// Core §6.8 — THE provided step-chain base: an SFC/ST/LD sequence POU extends
// this and gets the step record, condition waits, run-style pacing, the child
// PLCopen drive, delays, and the shared transition result — without re-declaring
// host plumbing per chain. The derived chart's actions are the only writers of
// _retVal; every chart transition reads it; one shared exit action calls
// M_ClearTransition. Framework flow-control lives here ONCE (§6.8(a)); the
// application's command/wait/decision logic stays visible in each step action.
FUNCTION_BLOCK ABSTRACT FB_SequenceBase IMPLEMENTS I_Sequence
VAR_OUTPUT
    ActiveStep : INT;              // §6.5 mirror of the step record (chart-local view)
    Done : BOOL;                   // finite chains: TRUE at their finish step
END_VAR
VAR
    _step    : INT;                // §6.5 active step index (the ST `CASE _step OF` token)
    // Shared transition result (§6.10). ONE-SCAN signal: the active step's action
    // is its only writer, every chart transition reads it, and it is cleared before
    // the next scan's actions run - by M_Advance on commit in an ST chart, or by
    // M_BeginScan when the chart runtime owns the transition (SFC/LD/FBD).
    _retVal  : E_StepResult;
    // §6.12 — the same one-scan signal as _retVal, but one per CONCURRENT LEG.
    // A parallel divergence has several active steps at once, so a single shared
    // result cannot work: whichever leg wrote last would decide every leg's
    // transition. Index n belongs to leg n; the main line keeps _retVal, so a
    // chain with no parallel branch never touches this array.
    //
    // A leg's step action writes `_conRetVal[n] := E_StepResult.ADVANCE;` and its
    // transition reads `_conRetVal[n] = E_StepResult.ADVANCE`; the join reads every
    // leg plus the main line. Cleared with _retVal once per scan (M_BeginScan), and
    // per leg on that leg's step exit (M_ClearTransition) - never across legs,
    // which would let one leg's commit erase another's result mid-motion.
    _conRetVal  : ARRAY[1..PL_Fraktal.MAX_PARALLEL_BRANCHES] OF E_StepResult;
    _restart : BOOL;               // a step may request a chart restart (M_Run applies it)
    {attribute 'OPC.UA.DA' := '0'}
    _host : I_SequenceHost;        // owning module's framework services (§6.7)
    _attached : BOOL;
    // §6.12 — every STEP-scoped latch is per CONCURRENT BRANCH, because two legs of
    // a parallel divergence are two active steps in the same POU at the same time.
    // Sharing one latch let leg A's issue consume leg B's, and let leg A's step exit
    // wipe leg B's transition result. Index 0 is the main line, which is what a chain
    // without any parallel branch uses throughout.
    _delay : ARRAY[0..PL_Fraktal.MAX_PARALLEL_BRANCHES] OF TON;
    _driveIssued : ARRAY[0..PL_Fraktal.MAX_PARALLEL_BRANCHES] OF BOOL;
    _subRunning : ARRAY[0..PL_Fraktal.MAX_PARALLEL_BRANCHES] OF BOOL;
    // Which leg the step action executing RIGHT NOW belongs to. Set by M_Step from
    // its `Branch` input, so it is always in step with the record just published,
    // and reset to _branchBase every scan - a chain that never names a leg is
    // therefore always on its own, which for a top-level chain is the main line.
    _branch : INT;
    // This chain's own leg index when the chain IS a leg (assigned by M_RunPar at
    // the fork). 0 for a top-level chain. It is what lets a leg written as its own
    // chain tag every one of its rows without naming a branch anywhere.
    _branchBase : INT;
    _lastStep : ARRAY[0..PL_Fraktal.MAX_PARALLEL_BRANCHES] OF INT;
    _stepSeen : ARRAY[0..PL_Fraktal.MAX_PARALLEL_BRANCHES] OF BOOL;
    _parStarted : ARRAY[1..PL_Fraktal.MAX_PARALLEL_BRANCHES] OF BOOL;
    _parLegs : INT;                // M_RunPar calls made this scan
    _parDone : INT;                // how many of them reported Done
    _errorRaised : BOOL;           // this chain raised the active fault (§6.9)
    _warnRaised : ARRAY[0..PL_Fraktal.MAX_PARALLEL_BRANCHES] OF BOOL;   // §6.9(e) one message per step visit
    _baseStepNo : INT;             // §6.5 step-record offset when run as a sub-chain
END_VAR

;

// §6.8 ST-skeleton progression: at the END of a `CASE _step OF` body, commit the
// step's shared transition result. On ADVANCE (or a declared JUMPn) go to the
// mapped next step and clear the step-scoped latches so the new step re-arms — the
// exact guarantee the SFC exit action gave, in one call. NONE stays put. The caller
// passes its successor map; an unmapped result holds the step (safe, visible).
METHOD M_Advance
VAR_INPUT
    OnAdvance : INT;               // next step for E_StepResult.ADVANCE
    // Jump targets default to "not used" so the common case reads
    // `M_Advance(OnAdvance := 100);` instead of repeating `OnJump1..3 := -1`.
    // Defaulted METHOD inputs need TwinCAT >= 3.1.4026, so on the legacy 4024
    // target (FRAKTAL_TC3_4024 defined) they are declared without defaults and
    // every argument is passed explicitly. See Params/PL_FraktalCompat.TcGVL.
    {IF defined (FRAKTAL_TC3_4024)}
    OnJump1   : INT;               // next step for JUMP1 (-1 = not used)
    OnJump2   : INT;               // next step for JUMP2 (-1 = not used)
    OnJump3   : INT;               // next step for JUMP3 (-1 = not used)
    {ELSE}
    OnJump1   : INT := -1;         // next step for JUMP1 (-1 = not used)
    OnJump2   : INT := -1;         // next step for JUMP2 (-1 = not used)
    OnJump3   : INT := -1;         // next step for JUMP3 (-1 = not used)
    {END_IF}
END_VAR
VAR
    target : INT;
END_VAR
target := -1;
CASE _retVal OF
    E_StepResult.ADVANCE: target := OnAdvance;
    E_StepResult.JUMP1:   target := OnJump1;
    E_StepResult.JUMP2:   target := OnJump2;
    E_StepResult.JUMP3:   target := OnJump3;
END_CASE
IF target >= 0 THEN
    _step := target;
    ActiveStep := target;
    M_ClearTransition();           // §6.10: a completed result never leaks into the next step
END_IF
END_METHOD

// §6.11 forward
METHOD M_AskDecision
VAR_INPUT
    Req : ST_DecisionRequest;
END_VAR
IF _host <> 0 THEN
    _host.M_SequenceAskDecision(Req := Req);
END_IF
END_METHOD

// bind the owner's host bridge; the derived Setup adds its typed child bindings.
METHOD M_Attach : BOOL
VAR_INPUT
    Host : I_SequenceHost;
END_VAR
_host := Host;
_attached := (Host <> 0);
IF _attached THEN
    // Announce this chain to its owner so the Unit base can run the
    // §6.10 per-scan result reset for it. The project writes nothing (O1).
    _host.M_SequenceRegister(Seq := THIS^);
END_IF
M_Attach := _attached;
END_METHOD

// §6.9(b) named plain-condition wait (forward to the host).
METHOD M_Await : BOOL
VAR_INPUT
    Idx : INT;
    Label : STRING(120);
    Ok : BOOL;
END_VAR
M_Await := FALSE;
IF _host <> 0 THEN
    M_Await := _host.M_SequenceAwait(Idx := Idx, Label := Label, Ok := Ok);
END_IF
END_METHOD

// Core §6.10 - scan-scoped reset of the shared transition result.
//
// `_retVal` is a ONE-SCAN signal: the active step's action writes it, the chart's
// transition reads it in the same scan, and it must not survive into the next.
// In an ST chart M_Advance is itself the transition, so it commits and clears in
// one call. In a chart language the RUNTIME evaluates transitions (SFC/LD/FBD),
// so nothing in the chart is positioned to clear afterwards - call this once per
// PLC cycle immediately BEFORE executing the chart. Clearing at the top of the
// scan is equivalent to clearing after the previous scan's transitions, and it
// forces every step action to re-assert its own result each scan, which is the
// property that makes a stale ADVANCE impossible.
//
// It deliberately clears ONLY the result. `_driveIssued` (M_TryIssue's one-shot)
// and `_delay` (M_Delay's timer) are STEP-scoped, not scan-scoped: resetting them
// every scan would re-issue a child command every cycle and stop any delay from
// ever elapsing. Those re-arm on step change, through M_ClearTransition.
METHOD M_BeginScan
VAR
	Idx : INT;
END_VAR
_retVal := E_StepResult.NONE;
FOR Idx := 1 TO PL_Fraktal.MAX_PARALLEL_BRANCHES DO
    _conRetVal[Idx] := E_StepResult.NONE;
END_FOR
// §6.12 the branch cursor is scan-scoped: a step action that does not declare a
// branch is on the main line (or on this chain's own leg when it IS a leg), so a
// chain with no parallel branch never mentions one.
_branch := _branchBase;
_parLegs := 0;
_parDone := 0;
END_METHOD

// Restart this chain as a sub-chain of a composite step: its step records are
// offset by the owning step number (§6.5) so the stall walk still reports one
// continuous chain. OnChainReset carries any application state.
METHOD M_ChainReset
VAR_INPUT
    BaseStepNo : INT;
    // §6.12 the leg index this chain runs as, assigned by the fork. 0 = not a leg.
    // Every step it records is tagged with it, so the project writes it once per
    // leg instead of once per step (§1.1 O1).
    Branch : INT;
END_VAR
_baseStepNo := BaseStepNo;
_branchBase := Branch;
M_ResetBase(FirstStep := 0);
OnChainReset();
END_METHOD

// §6.12 — the join of a parallel step: ADVANCE on the scan every leg run this
// scan has reported Done, NONE while any is still working. The counts are
// scan-scoped, so the join always reflects the legs the step actually ran -
// there is no leg list to register, and none to forget to update (§1.1 O1).
METHOD M_ParJoin : E_StepResult
M_ParJoin := E_StepResult.NONE;
IF (_parLegs > 0) AND (_parDone = _parLegs) THEN
    M_ParJoin := E_StepResult.ADVANCE;
END_IF
END_METHOD

// §6.12 — run one leg of a parallel step. THE portable form of a parallel
// divergence, and the only one available to an ST chain.
//
//     M_Step(StepNo := 500, StepName := 'project.step.bothPositions', ...);
//     M_RunPar(Chain := _positionA, BaseStepNo := 500, Branch := 1);
//     M_RunPar(Chain := _positionB, BaseStepNo := 600, Branch := 2);
//     _retVal := M_ParJoin();
//     M_Advance(OnAdvance := 999);
//
// Each leg is an ordinary FB_SequenceBase chain, so it brings its own step
// pointer, its own transition result and its own step-scoped latches - the
// collisions §6.12 has to manage inside one POU simply cannot arise (§1.1 O4:
// the model scales structurally rather than by decoration). Its steps are
// recorded under BaseStepNo and tagged with Branch, so the §3.13 flow chart
// groups them and the §6.9 walk still names one continuous chain.
//
// Returns TRUE on the scans this leg reports Done. The entry latch is
// step-scoped, so re-entering the fork step later restarts every leg.
METHOD M_RunPar : BOOL
VAR_INPUT
    Chain : REFERENCE TO FB_SequenceBase;
    BaseStepNo : INT;
    Branch : INT;
END_VAR
M_RunPar := FALSE;
IF NOT __ISVALIDREF(Chain) THEN
    RETURN;
END_IF
IF (Branch < 1) OR (Branch > PL_Fraktal.MAX_PARALLEL_BRANCHES) THEN
    M_Fault(Reason := E_Reason.UNSUPPORTED_COMMAND,
        DescriptionKey := 'std.error.parallelBranchOutOfRange');
    RETURN;                          // §5.6 no silent default
END_IF
IF NOT _parStarted[Branch] THEN
    Chain.M_ChainReset(BaseStepNo := BaseStepNo, Branch := Branch);
    _parStarted[Branch] := TRUE;
END_IF
Chain.M_ChainRun();
_parLegs := _parLegs + 1;
IF Chain.Done THEN
    _parDone := _parDone + 1;
    M_RunPar := TRUE;
END_IF
END_METHOD

// One scan of this chain. An ST chart overrides this with its
// `CASE _step OF` body; a chart-language POU leaves it alone because its own body
// IS the chart and the runtime executes it. Only a chain that is used as a
// composite step (M_RunSub) has to override it.
METHOD M_ChainRun
;
END_METHOD

METHOD M_ClearDecision
IF _host <> 0 THEN
    _host.M_SequenceClearDecision();
END_IF
END_METHOD

// the ONE shared STEP-EXIT action: a completed step's result never leaks into
// the next step, and the step-scoped helpers (delay, drive latch) re-arm.
// §6.12 — it re-arms THE CURRENT BRANCH only. Clearing every branch here is what
// made a parallel divergence misbehave: one leg committing a step wiped the other
// leg's transition result and its issue latch mid-motion.
// ST charts reach this through M_Advance on commit. A chart language whose
// engine owns the transition (SFC/LD/FBD) wires this as the step exit action,
// which the runtime executes AFTER the transition condition was evaluated -
// so the transition still sees the result the step action produced.
METHOD M_ClearTransition
VAR
	Idx : INT;
END_VAR
IF _branch = 0 THEN
    _retVal := E_StepResult.NONE;
    // A fork always sits on the main line of its own chain (§6.12), so leaving the
    // fork step is what re-arms its legs for a later re-entry.
    FOR Idx := 1 TO PL_Fraktal.MAX_PARALLEL_BRANCHES DO
        _parStarted[Idx] := FALSE;
    END_FOR
ELSE
    _conRetVal[_branch] := E_StepResult.NONE;
END_IF
_driveIssued[_branch] := FALSE;
_warnRaised[_branch] := FALSE;
_subRunning[_branch] := FALSE;
_delay[_branch](IN := FALSE);
END_METHOD

// §6.1 one-shot completion forward (finite chains)
METHOD M_Complete
IF _host <> 0 THEN
    _host.M_SequenceComplete();
END_IF
END_METHOD

METHOD M_CountGood
IF _host <> 0 THEN
    _host.M_SequenceCountGood();
END_IF
END_METHOD

// a declared process wait in ONE step (settle/dwell). The timer runs while the
// step is active and re-arms through the shared exit action.
METHOD M_Delay : E_StepResult
VAR_INPUT
    PT : TIME;
END_VAR
M_Delay := E_StepResult.NONE;
_delay[_branch](IN := TRUE, PT := PT);
IF _delay[_branch].Q THEN
    _delay[_branch](IN := FALSE);
    M_Delay := E_StepResult.ADVANCE;
END_IF
END_METHOD

// §8.11.1 cycle-complete marker forward; FALSE = stop granted (do not loop)
METHOD M_EndOfCycle : BOOL
M_EndOfCycle := FALSE;
IF _host <> 0 THEN
    M_EndOfCycle := _host.M_SequenceEndOfCycle();
END_IF
END_METHOD

// §6.9 first-out fault from a step (forward to the host).
METHOD M_Fault
VAR_INPUT
    Reason : E_Reason;
    DescriptionKey : STRING(255);
END_VAR
IF _host <> 0 THEN
    _host.M_SequenceFault(Reason := Reason, DescriptionKey := DescriptionKey);
END_IF
END_METHOD

// §3.4.2 run-style pacing gate (forward to the host).
METHOD M_Gate : BOOL
VAR_INPUT
    Steppable : BOOL;
END_VAR
M_Gate := FALSE;
IF _host <> 0 THEN
    M_Gate := _host.M_SequenceStepGate(Steppable := Steppable);
END_IF
END_METHOD

// §6.1 issue+await in ONE step: TRUE exactly once per step visit, when the
// run-style gate permits (§3.4.2). The action then sets the child's typed
// Command and raises Execute — visibly, in the step (§6.8). The child's Done
// releases the handshake and sets _retVal := ADVANCE; a child Error needs no
// step code — the owning Unit adopts it instantly via the §8.2 rollup.
// The latch re-arms through the shared exit action (M_ClearTransition).
METHOD M_TryIssue : BOOL
VAR_INPUT
    Steppable : BOOL;
END_VAR
M_TryIssue := FALSE;
IF _driveIssued[_branch] THEN
    RETURN;
END_IF
IF M_Gate(Steppable := Steppable) THEN
    _driveIssued[_branch] := TRUE;
    M_TryIssue := TRUE;
END_IF
END_METHOD

METHOD M_PartProcessed : BOOL
VAR_INPUT
    Verdict : E_Verdict;
    Reason : E_Reason;
END_VAR
M_PartProcessed := FALSE;
IF _host <> 0 THEN
    M_PartProcessed := _host.M_SequencePartProcessed(Verdict := Verdict, Reason := Reason);
END_IF
END_METHOD

// §3.16.3 forward (framework plumbing stays out of step actions).
METHOD M_PartReceived : BOOL
M_PartReceived := FALSE;
IF _host <> 0 THEN
    M_PartReceived := _host.M_SequencePartReceived();
END_IF
END_METHOD

METHOD M_PartRecord : BOOL
VAR_INPUT
    RecordName : STRING(64);
    Value : LREAL;
    Minimum : LREAL;
    Maximum : LREAL;
    Target : LREAL;
    EngUnit : STRING(16);
END_VAR
M_PartRecord := FALSE;
IF _host <> 0 THEN
    M_PartRecord := _host.M_SequencePartRecord(RecordName := RecordName,
        Value := Value, Minimum := Minimum, Maximum := Maximum, Target := Target,
        EngUnit := EngUnit);
END_IF
END_METHOD

METHOD M_PartStarted
IF _host <> 0 THEN
    _host.M_SequencePartStarted();
END_IF
END_METHOD

// §6.9/§8.8 — raise a message this step defines itself.
//
// For a condition the framework cannot see: a measured value out of band, a
// disagreement between two children, an application rule. LinkPath is the module
// the §3.13 chart should drill into ('' = this Unit).
//
// Severity and Category are a PROPOSAL, not the last word: adoption runs the §8.8
// rationalization, so a reason that is in the registry gets the registry's priority
// and category and these inputs are ignored. They survive for a project band code
// (10000+) the registry does not know - which is exactly where a custom message of
// a different level belongs.
METHOD M_RaiseCustom : BOOL
VAR_INPUT
    Reason         : E_Reason;
    DescriptionKey : STRING(255);
    Severity       : E_Severity;
    Category       : E_Category;
    LinkPath       : STRING(255);
END_VAR
VAR
    diag : ST_Diagnostic;
END_VAR
M_RaiseCustom := FALSE;
IF _host = 0 THEN
    RETURN;
END_IF
diag.ReasonCode  := Reason;
diag.Description := DescriptionKey;
diag.SourcePath  := LinkPath;
diag.Severity    := Severity;
diag.Category    := Category;
M_RaiseCustom := _host.M_SequenceRaise(Diag := diag, LinkPath := LinkPath);
_errorRaised := M_RaiseCustom;
END_METHOD

// §6.9 — adopt a child's first-out from inside conditional step logic.
//
// `Awaits` rolls a child fault up automatically, but only for a step that hands
// the child to the framework. A step that decides for itself - anything with an
// IF or CASE around the command - calls this instead, and gets the same result:
// the child's reason verbatim, the child's path as the §3.13 drill-down link,
// and the chain stopped until the error is cleared.
//
// Returns TRUE only when a fault was actually raised, so the usual shape is
//     IF M_RaiseFromChild(Source := _pressRam) THEN RETURN; END_IF
METHOD M_RaiseFromChild : BOOL
VAR_INPUT
    Source : I_Module;
END_VAR
M_RaiseFromChild := FALSE;
IF Source = 0 THEN
    RETURN;
END_IF
IF NOT Source.FaultActive THEN
    RETURN;                          // nothing to raise: safe to call every scan
END_IF
IF _host = 0 THEN
    RETURN;
END_IF
M_RaiseFromChild := _host.M_SequenceRaise(Diag := Source.GetFaultSummary(),
    LinkPath := Source.Name);
_errorRaised := M_RaiseFromChild;
END_METHOD

// §6.9(e) — a custom message that informs and lets the chain carry on.
//
// For designed behaviour with a consequence worth recording: an operator
// releasing a two-hand control mid-motion, a retry, a value drifting inside its
// band. It is NOT the error path - the chain is not stopped, no fault is
// adopted, and the step keeps whatever recovery it already routes to.
//
// Raised at most ONCE per visit to a step, however many scans the step runs and
// however many times this is called (§1.1 O1: a project shall never have to
// remember an edge latch for correctness). Committing the step re-arms it.
//
// Severity/Category are the caller's for a project band code; a reason in the
// §8.8 registry is rationalized to the registry's values like any other.
METHOD M_RaiseWarning : BOOL
VAR_INPUT
    Reason         : E_Reason;
    DescriptionKey : STRING(255);
    Severity       : E_Severity;
    Category       : E_Category;
END_VAR
VAR
    diag : ST_Diagnostic;
END_VAR
M_RaiseWarning := FALSE;
IF _warnRaised[_branch] OR (_host = 0) THEN
    RETURN;                          // already said once for this visit
END_IF
diag.ReasonCode  := Reason;
diag.Description := DescriptionKey;
diag.Severity    := Severity;
diag.Category    := Category;
M_RaiseWarning := _host.M_SequenceWarn(Diag := diag);
_warnRaised[_branch] := M_RaiseWarning;
END_METHOD

// §6.9(e) — publish a child's failure WITHOUT adopting it.
//
// The counterpart of M_RaiseFromChild, for a step that already owns the
// recovery: the child's first-out reaches the alarm ring and the §3.13 chart
// (marked on this step, click-through to the child), but nothing faults and the
// chain keeps the branch it was going to take anyway. Press AUTO N200 is the
// case: the ram not reaching is handled by an operator confirmation and a scrap,
// so stopping there would replace a designed recovery with a hard fault - while
// saying nothing left the failure invisible on the Unit.
//
// Reported once per visit to the step, so calling it every scan is correct.
METHOD M_ReportFromChild : BOOL
VAR_INPUT
    Source : I_Module;
END_VAR
M_ReportFromChild := FALSE;
IF _warnRaised[_branch] OR (_host = 0) OR (Source = 0) THEN
    RETURN;
END_IF
IF NOT Source.FaultActive THEN
    RETURN;                          // nothing to report: safe every scan
END_IF
M_ReportFromChild := _host.M_SequenceWarn(Diag := Source.GetFaultSummary());
_warnRaised[_branch] := M_ReportFromChild;
END_METHOD

// clear the base flow state to the first step. The derived M_Reset calls this.
METHOD M_ResetBase
VAR_INPUT
    // Defaults to 0 (N000), the conventional first step, so a derived M_Reset
    // reads `M_ResetBase();`. Legacy 4024 has no defaulted method inputs, so
    // there the argument is required — see Params/PL_FraktalCompat.TcGVL.
    {IF defined (FRAKTAL_TC3_4024)}
    FirstStep : INT;               // the chain's initial step number (N000 = 0)
    {ELSE}
    FirstStep : INT := 0;          // the chain's initial step number (N000 = 0)
    {END_IF}
END_VAR
VAR
    Idx : INT;
END_VAR
_step := FirstStep;
ActiveStep := FirstStep;
Done := FALSE;
_restart := FALSE;
// §6.12 a reset re-arms EVERY branch, not just the one that happened to run last.
FOR Idx := 0 TO PL_Fraktal.MAX_PARALLEL_BRANCHES DO
    _stepSeen[Idx] := FALSE;
    _lastStep[Idx] := -1;
    _branch := Idx;
    M_ClearTransition();
END_FOR
_branch := _branchBase;
_parLegs := 0;
_parDone := 0;
END_METHOD

// §6.8 I_Sequence - start over at N000 with the chain's own state cleared. The
// owning Unit calls this for every attached chain on first scan, mode change and
// both abort paths, and a project calls it (through _M_RestartSequences) where
// its own restart-or-resume policy says so. A chain puts the state it owns in
// OnChainReset and writes no reset method of its own (§1.1 O1).
METHOD M_Restart
M_ResetBase(FirstStep := 0);
OnChainReset();
END_METHOD

// §6.9 — the owning Unit left ERROR. The chain's _step was never touched, so it
// resumes exactly where it stopped; re-arming the step-scoped latches here is
// what makes it RE-EVALUATE the command rather than resume mid-handshake with a
// spent M_TryIssue one-shot and a half-run delay.
METHOD M_ResumeAfterError
IF NOT _errorRaised THEN
    RETURN;
END_IF
_errorRaised := FALSE;
M_ClearTransition();
END_METHOD

// §6.8 run another chain as ONE composite step. Returns NONE while the
// sub-chain works and ADVANCE on the scan it finishes, so a step action reads:
//
//     _retVal := M_RunSub(Chain := _loadPosition, BaseStepNo := 240);
//
// The entry latch is step-scoped and re-arms through M_ClearTransition, so a
// chain re-entered later restarts correctly. The sub-chain inherits the leg of
// the step that runs it (§6.12), so a composite step inside a parallel branch
// publishes its sub-steps under that leg without saying so. Hand-written, this was eight lines
// per composite step and one forgotten latch reset left a chain that never ran
// again (§1.1 O1: the framework owns repeated flow control, not the project).
METHOD M_RunSub : E_StepResult
VAR_INPUT
    Chain : REFERENCE TO FB_SequenceBase;
    BaseStepNo : INT;
END_VAR
M_RunSub := E_StepResult.NONE;
IF NOT __ISVALIDREF(Chain) THEN
    RETURN;
END_IF
IF NOT _subRunning[_branch] THEN
    // §6.12 — the sub-chain runs INSIDE this step, so it belongs to whatever leg
    // this step is on. _branch is already correct (M_Step set it from the step
    // record), so there is nothing for the project to state and nothing that can
    // drift out of step with the record - the same reason Branch is an input of
    // M_Step rather than a call beside it (§1.1 O1).
    Chain.M_ChainReset(BaseStepNo := BaseStepNo, Branch := _branch);
    _subRunning[_branch] := TRUE;
END_IF
Chain.M_ChainRun();
IF Chain.Done THEN
    _subRunning[_branch] := FALSE;
    M_RunSub := E_StepResult.ADVANCE;
END_IF
END_METHOD

// §6.5 step record + the chart-local ActiveStep mirror, one call.
METHOD M_Step
VAR_INPUT
    StepNo : INT;
    StepName : STRING(120);
    Awaits : I_Module;
    AwaitingLabel : STRING(120);
    TimeClass : E_TimeClass;
    ExpectedTime : TIME;
    // §6.12 — the concurrent leg this step belongs to, which a step on the main
    // line never mentions. Folding it into the step record rather than a separate
    // call is what makes it impossible to declare a leg without recording a step,
    // or to record a step under the wrong leg because the declaration was
    // forgotten (§1.1 O1: the framework owns the bookkeeping, not the project).
    // 0 means "this chain's own leg", which is the main line for a top-level chain
    // and the index the fork assigned for a chain running as a leg (M_RunPar) -
    // so a leg written as its own chain never mentions a branch either.
    {IF defined (FRAKTAL_TC3_4024)}
    Branch : INT;
    {ELSE}
    Branch : INT := 0;
    {END_IF}
END_VAR
// §6.12 — select the leg first: everything below, and everything the step action
// does after this call (M_TryIssue, M_Delay, M_RunSub, the §6.9(e) message latch)
// is scoped to it. An out-of-range index faults rather than quietly landing on the
// main line (§5.6 - no silent default).
IF Branch < 0 OR Branch > PL_Fraktal.MAX_PARALLEL_BRANCHES THEN
    M_Fault(Reason := E_Reason.UNSUPPORTED_COMMAND,
        DescriptionKey := 'std.error.parallelBranchOutOfRange');
    RETURN;
END_IF
IF Branch > 0 THEN
    _branch := Branch;
ELSE
    _branch := _branchBase;
END_IF
// A chart language never calls M_ClearTransition: its engine owns the transition,
// so there is no commit point to hang it on. The step record is the one call every
// step of every language makes, so the re-arm belongs here - a new step number on
// this leg re-arms that leg's issue latch, delay and message. Without it
// M_TryIssue fired once per chart RUN instead of once per step.
IF (NOT _stepSeen[_branch]) OR (_lastStep[_branch] <> StepNo) THEN
    _lastStep[_branch] := StepNo;
    _stepSeen[_branch] := TRUE;
    M_ClearTransition();
END_IF
ActiveStep := StepNo;
IF _host <> 0 THEN
    _host.M_SequenceSetStep(StepNo := StepNo, StepName := StepName, Awaits := Awaits,
        AwaitingLabel := AwaitingLabel, TimeClass := TimeClass, ExpectedTime := ExpectedTime,
        Branch := _branch);
END_IF
END_METHOD

// §3.4/§8.11 — accept the stop between cycles (forward to the host).
METHOD M_StopNow
IF _host <> 0 THEN
    _host.M_SequenceStopNow();
END_IF
END_METHOD

// §3.4 — poll at the between-cycles wait step (forward to the host).
METHOD M_StopPending : BOOL
M_StopPending := FALSE;
IF _host <> 0 THEN
    M_StopPending := _host.M_SequenceStopPending();
END_IF
END_METHOD

METHOD M_TakeDecision : INT
M_TakeDecision := 0;
IF _host <> 0 THEN
    M_TakeDecision := _host.M_SequenceTakeDecision();
END_IF
END_METHOD

// §3.14 hook: clear application-owned chain state on restart. Empty by default
// so a chain that has none writes nothing.
METHOD PROTECTED OnChainReset
;
END_METHOD

END_FUNCTION_BLOCK

(* stored: Version 1.1.0.1
   POU FB_SequenceBase: Id {6c2f91a4-3e87-4b5d-a1f0-58d24c7be093}, SpecialFunc None
   Method M_Advance: Id {a71c4d38-52e9-4b06-9f81-3d0e6c25a704}
   Method M_AskDecision: Id {c60f93b2-1e78-4ad5-8b40-97d2e5c1a083}
   Method M_Attach: Id {83d17f5a-2b64-4c09-9ae8-01f6b2d47c35}
   Method M_Await: Id {7d05e9c3-46a2-4f81-92b6-e3157cd80a49}
   Method M_BeginScan: Id {4c0862c1-7015-4c44-8473-90c09e6eebff}
   Method M_ChainReset: Id {a41025db-fb80-43ee-99ef-bace7f63f844}
   Method M_ParJoin: Id {f98ae9d3-390d-46f9-904f-3a62bb18f212}
   Method M_RunPar: Id {707c763b-a5d2-4ecb-bf74-ae809dae7fd3}
   Method M_ChainRun: Id {b2dd28b6-7db9-48a6-8f4e-a437e83baa79}
   Method M_ClearDecision: Id {4b06d8e1-72af-4c95-a3d8-e50c19b7f234}
   Method M_ClearTransition: Id {2e6b48d1-95cf-4a73-b30e-6f81da29c504}
   Method M_Complete: Id {68e5b09c-d3f1-4a27-85b6-04c7a2e91d58}
   Method M_CountGood: Id {31d84e0a-6cf2-49b7-90e5-2af7c81d53b6}
   Method M_Delay: Id {e94b06d2-571c-4a88-9fe3-c07a35d21b60}
   Method M_EndOfCycle: Id {d95f31a8-40c6-4e7b-92d0-6b18e4c5f7a9}
   Method M_Fault: Id {0b83f5e7-92c6-4d1a-8f40-56a91dce27b8}
   Method M_Gate: Id {49c8e2b7-1af3-4d50-a6e9-8b02f47c9d16}
   Method M_TryIssue: Id {d70a5c94-83e1-4f26-b5d8-42c69e01af37}
   Method M_PartProcessed: Id {9f5a2c18-b7e4-4063-a58d-1e6c30d9f427}
   Method M_PartReceived: Id {7c3e0f91-2ab8-4d64-95c7-e8140b6a25d9}
   Method M_PartRecord: Id {e21b7f60-93d5-4a8c-8f14-c5d09e3b7a42}
   Method M_PartStarted: Id {5d19c4a7-8e02-4f5b-b6d3-70f28c1e94a6}
   Method M_RaiseCustom: Id {11030a2b-446d-408a-be8e-77b2d821a339}
   Method M_RaiseFromChild: Id {df83c77d-bc83-42e1-ac7d-6193bc3a0362}
   Method M_RaiseWarning: Id {3fe15fab-e9b5-4d06-9baf-f8b35615c629}
   Method M_ReportFromChild: Id {3c0625b4-1691-42a6-8198-5d21de9ddfe5}
   Method M_ResetBase: Id {5a90c3e2-7f18-4d66-8b2a-9ce45d10f782}
   Method M_Restart: Id {79b49099-977a-4b6b-a0e0-49fea2634ec6}
   Method M_ResumeAfterError: Id {60fcb1e5-ca9a-42a5-8f04-39fe8ddf26c0}
   Method M_RunSub: Id {c441a4bf-6a3a-473d-aecf-8dcf381358dc}
   Method M_Step: Id {b1f42a68-0d95-4e37-8cb1-27d3a9e60f14}
   Method M_StopNow: Id {1a97d3c8-45e2-4bf1-8d06-b52c8fe0a374}
   Method M_StopPending: Id {f6c14e29-8b70-4da3-95c2-30e8a1d7f465}
   Method M_TakeDecision: Id {a84c17f5-05d9-4e32-b6a1-38f0c92d67e4}
   Method OnChainReset: Id {6e368c40-f3a8-46a7-866a-7e436102e0a9} *)
